(* LS Electric XG5000 project: 241008_연습문제9 *)
(* PLC LSPLC *)

PROGRAM NewProgram (* task: 스캔 프로그램 *)
VAR
    P1 AT %IX0.0.0 : BOOL;
    P10 AT %QX0.1.0 : BOOL;
    P11 AT %QX0.1.1 : BOOL;
    P12 AT %QX0.1.2 : BOOL;
    T1 : TON;
    T2 : TON;
    T3 : TON;
    내부메모리 AT %MX0 : BOOL;
END_VAR

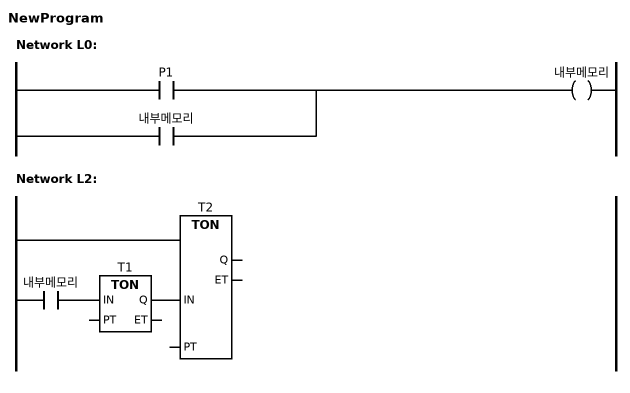
(* Rung L0 *)
내부메모리 := P1 OR 내부메모리;
(* Rung L2 *)
T1(IN := 내부메모리);
T2(IN := T1.Q);
END_PROGRAM